FUNCTION "IPC_Push_Log_MES" : Void
{ S7_Optimized_Access := 'TRUE' ; Published := 'FALSE' }
VERSION : 0.1
   VAR_INPUT
      Msg : "MES_Msg";
      Ack : DInt;
   END_VAR

   VAR_TEMP
      RETVAL : Int;
   END_VAR


BEGIN

	(*
	recupera l'ultimo messaggio inviato a MES = messaggio topic = 101

	#""MES_Send_Buffer_Msg_Topic1XX".msg[0]"

	*)
	;




END_FUNCTION

